Staubli VAL3: insertInstr.pgx

program insertInstr(InstrItem& x_iItem[])
  local num i
  local num l_nIndex
  local string l_sPath
  local string l_sItem
begin
  // TODO
  call use:setSizeList(14,0,10,11)
  call use:setView(false)
  call use:listcreate("Select")
  // insert the action on Point
  call use:listadd(saveData:sInstrOnPoint)
  call use:listupdate(0)
  // SELECT THE ITEM
  do
    i=get()
    call use:listevent(i,l_nIndex,l_sItem)
  until i==255 or i==270
  // copy
  x_iItem.sType=l_sItem
  // define it
  if x_iItem.sType!="" and i==270
    // load the instruction
    call saveData:getPathInstr(x_iItem.sType,l_sPath)
    // load the instruction
    events:libLoad(l_sPath)
    delay(0)
    call events:onInsert(x_iItem.sData)
    // insert the item
    return
  endIf
  // NOT GOOD
  x_iItem.sType=""
  x_iItem.sData=""
end
